FUNCTION_BLOCK PUBLIC TmsExchange EXTENDS Process
VAR
	_TmsSwitch : ITF_TmsSwitch;
	_StateMachine : IPmlStateMachine;
	
	embarkingStation : TmsEmbarkStation := (BoardVelocity := 100.0);
	holdingStation : TmsHoldStation := (MyEmbarkStation := embarkingStation);
END_VAR

{analysis -2}

PROPERTY BoardingVelocity : MC_LREAL
GET
BoardingVelocity := embarkingStation.BoardVelocity;
END_GET
SET
embarkingStation.BoardVelocity := BoardingVelocity;
END_SET
END_PROPERTY

METHOD PUBLIC  Cycle : HRESULT
VAR
END_VAR
Cycle := holdingStation.Cycle();
Cycle := embarkingStation.Cycle();
END_METHOD

PROPERTY EmbarkStation : IProcess
GET
EmbarkStation := embarkingStation;
END_GET
END_PROPERTY

PROPERTY ExchangePosition : MC_LREAL
GET
END_GET
SET
embarkingStation.Position := ExchangePosition + 150;
holdingStation.Position := ExchangePosition;
END_SET
END_PROPERTY

PROPERTY ExchangeTrackLevel : int
GET
ExchangeTrackLevel := embarkingStation.TrackLevel;
END_GET
SET
embarkingStation.TrackLevel := ExchangeTrackLevel;
END_SET
END_PROPERTY

PROPERTY HoldStation : IProcess
GET
HoldStation := holdingStation;
END_GET
END_PROPERTY

PROPERTY MyStateMachine : IPmlStateMachine
GET
MyStateMachine := _StateMachine;
END_GET
SET
_StateMachine := MyStateMachine;
embarkingStation.MyStateMachine := MyStateMachine;
holdingStation.MyStateMachine := MyStateMachine;
END_SET
END_PROPERTY

PROPERTY SwitchTravelPosition : MC_LREAL
GET
SwitchTravelPosition := embarkingStation.SwitchTravelPosition;
END_GET
SET
embarkingStation.SwitchTravelPosition := SwitchTravelPosition;
END_SET
END_PROPERTY

PROPERTY TmsSwitch : ITF_TmsSwitch
GET
TmsSwitch := _TmsSwitch;
END_GET
SET
_TmsSwitch := TmsSwitch;
embarkingStation.TmsSwitch := TmsSwitch;
END_SET
END_PROPERTY

PROPERTY PUBLIC TrackIds : Array[1..4] of OTCID
GET
TrackIds := embarkingStation.TrackIds;
END_GET
SET
embarkingStation.TrackIds := TrackIds;
END_SET
END_PROPERTY

END_FUNCTION_BLOCK

(* stored: Version 1.1.0.1, ProductVersion 3.1.4024.12
   POU TmsExchange: Id {bbb0a31b-f62e-4332-abc9-0bed198282f3}, SpecialFunc None
   Property BoardingVelocity: Id {f532572a-3453-4f92-ae10-30b70032b173}
   Get Get: Id {1407af9b-7f2d-4421-bc6a-f91e47db8760}
   Set Set: Id {b4a11e16-1037-43d0-a3b7-848b029a697b}
   Method Cycle: Id {90b295e7-21c8-4280-8b63-dc25678715c4}
   Property EmbarkStation: Id {508d1299-8885-4c14-a332-b33475d26bfa}
   Get Get: Id {ba314324-3359-4a1a-8fb3-9807e1185edd}
   Property ExchangePosition: Id {72e7b26a-6207-46b0-b684-ab389b8f74bf}
   Get Get: Id {42f393b6-25e0-471d-b60d-0c33ee8e8a32}
   Set Set: Id {274655bc-bc44-4815-a7c2-3b11c6090289}
   Property ExchangeTrackLevel: Id {416bdb5b-acd9-4922-a121-e2d3d8d0274e}
   Get Get: Id {7ed999f7-41f4-4d02-9f01-a951336030fa}
   Set Set: Id {8abbf63f-29fc-48f1-952c-afd65680f071}
   Property HoldStation: Id {4d40e862-480a-426f-89ed-edc013bb8c8d}
   Get Get: Id {7b1202a4-917f-403c-b005-ec2e639cb9d8}
   Property MyStateMachine: Id {4196edef-498e-4d46-b5a7-e2b4ce4210df}
   Get Get: Id {3b4361b8-6ce6-4b1e-8f45-beceafdcd3a9}
   Set Set: Id {37aebee1-03ef-4127-a412-f2661d8be0ba}
   Property SwitchTravelPosition: Id {81526570-b9a9-41d5-adf0-49b50e38e46c}
   Get Get: Id {cd5a599e-fb72-4d8d-b6d6-a8e1cee905ed}
   Set Set: Id {0719daf7-7733-4b8b-a540-a379e8bb6a64}
   Property TmsSwitch: Id {85a620f6-c211-4e12-b763-3ad2fed889bb}
   Get Get: Id {b943f30d-f4ed-4d81-b9a4-8eb6002901bc}
   Set Set: Id {cb3000c8-bad5-4070-9c48-eb4e16c736f9}
   Property TrackIds: Id {31a30eda-833a-450a-89f7-9d9f22e2b4ec}
   Get Get: Id {a5973870-9ace-4fb7-8902-58880a368a69}
   Set Set: Id {aaa19c3a-1ba5-4ce2-9f99-79124cbc0dbc} *)
